Universal Robots PolyScope program: GlobalToControl.urp

Program GlobalToControl (installation=Youssef directory=/programs/Youssef createdIn=5.9.5.1031259 lastSavedIn=5.9.5.1031259 robotSerialNumber=20215500597)
Calibrated DH parameters: a=[0.000193, -0.066673, -0.391568, -0.000012, 0.00005, 0]; d=[0.162643, -472.05677, 465.132521, 7.058239, 0.099746, 0.099582]; alpha=[1.571116, 0.00089, 0.003862, 1.569269, -1.569248, 0]; deltaTheta=[0, -1.413394, 7.628392, 0.068187, 0, -0.000001]
Robot Program (runOnlyOnce=true)
  MoveJ speed 60 deg/s, acceleration 80 deg/s^2 (useActiveTCP=true) feature=Base
    SafeHome (positionOptionType=SPEED_AND_ACCELERATION speed=1.047198 acceleration=1.396263 nextMotionTime=2)
    Waypoint Pre_Global: TCP in base x=424.817 y=-1.551 z=1080.554 mm, rx=-1.2067 ry=1.2116 rz=-1.2125 rad; joints [89.999, -90, 0, -89.996, -0.001, -0.002] deg; TCP offset x=0 y=0 z=191.5 mm, rx=0 ry=0 rz=0 rad
    URCap Gripper Activate (Robotiq_Grippers, Robotiq Inc.) dataModel(ResetAndActivateKey=false)
    URCap Gripper (Robotiq_Grippers, Robotiq Inc.) dataModel(position=100.0, force=0.0, speed=30.0, positionInDouble=100.0, forceInDouble=0.0, speedInDouble=30.0, slaveIds=[9], blocking=true)
    Waypoint Waypoint_2: TCP in base x=551.14 y=80.155 z=946.388 mm, rx=-1.3882 ry=1.5372 rz=-1.1084 rad; joints [175.158, -73.344, -0.017, -87.688, -91.199, -0.001] deg
    Waypoint Waypoint (Variable): variable(featureName=Control_Standby)
